PROGRAM Prg_Match
VAR
	
	boChoisirAction: BOOL;
	intChoixAction: INT;
	i: INT;
	intPrioMaxTrouvee: INT;
	boVerifPrerequis: BOOL;
	j: INT;
	intVerifAction: USINT;
	intNbActionVerifTot: INT;
	intNbActionVerifDone: INT;
	TON_1 : TON;
	boVerifPucAttente: BOOL;
	intNbPucsPris: INT;
	intNbPucDansRobot: INT;
	boGoldPris: BOOL;
	R_TRIG_StartMove: R_TRIG;
	R_TRIG_Depl: R_TRIG;
	R_TRIG_Algo: R_TRIG;
	TON_2: TON;
	R_TRIG_Move: R_TRIG;
	ADSREAD_1: ADSREAD;
	boResetExp : BOOL := TRUE;
	ADSWRITE_1: ADSWRITE;
	TON_Blink1: TON;
	TON_Blink2: TON;
	ADSWRITE_2: ADSWRITE;
	boDesactiverExp: BOOL := FALSE;;
	boEtatReset: BOOL;
	ADSREAD_2: ADSREAD;
	TON_reset: TON;
	R_TRIG_Etape: R_TRIG;
	NbPucsBalance: INT;
	bRenewDeplEv: BOOL;
	boLireEtatExp: BOOL;
	ADSREAD_3: ADSREAD;
	R_TRIG_Agold: R_TRIG;
	R_TRIG_APousser: R_TRIG;
	R_TRIG_Aok : R_TRIG;
	test: BOOL;
	attentefront: BOOL;
END_VAR

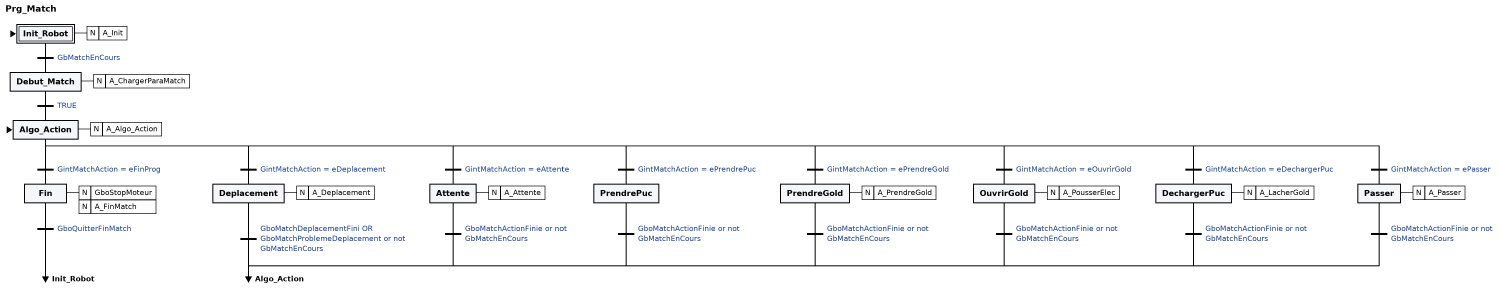
INITIAL_STEP Init_Robot:
    A_Init(N);
END_STEP
TRANSITION FROM Init_Robot TO Debut_Match
    := GbMatchEnCours;
END_TRANSITION
STEP Debut_Match:
    A_ChargerParaMatch(N);
END_STEP
TRANSITION FROM Debut_Match TO Algo_Action
    := TRUE;
END_TRANSITION
STEP Algo_Action:
    A_Algo_Action(N);
END_STEP
TRANSITION FROM Algo_Action TO Fin
    := GintMatchAction = eFinProg;
END_TRANSITION
STEP Fin:
    GboStopMoteur(N);
    A_FinMatch(N);
END_STEP
TRANSITION FROM Fin TO Init_Robot
    := GboQuitterFinMatch;
END_TRANSITION
TRANSITION FROM Algo_Action TO Deplacement
    := GintMatchAction = eDeplacement;
END_TRANSITION
STEP Deplacement:
    A_Deplacement(N);
END_STEP
TRANSITION FROM Deplacement TO Algo_Action
    := GboMatchDeplacementFini OR GboMatchProblemeDeplacement or not GbMatchEnCours;
END_TRANSITION
TRANSITION FROM Algo_Action TO Attente
    := GintMatchAction = eAttente;
END_TRANSITION
STEP Attente:
    A_Attente(N);
END_STEP
TRANSITION FROM Attente TO Algo_Action
    := GboMatchActionFinie or not GbMatchEnCours;
END_TRANSITION
TRANSITION FROM Algo_Action TO PrendrePuc
    := GintMatchAction = ePrendrePuc;
END_TRANSITION
STEP PrendrePuc:
END_STEP
TRANSITION FROM PrendrePuc TO Algo_Action
    := GboMatchActionFinie or not GbMatchEnCours;
END_TRANSITION
TRANSITION FROM Algo_Action TO PrendreGold
    := GintMatchAction = ePrendreGold;
END_TRANSITION
STEP PrendreGold:
    A_PrendreGold(N);
END_STEP
TRANSITION FROM PrendreGold TO Algo_Action
    := GboMatchActionFinie or not GbMatchEnCours;
END_TRANSITION
TRANSITION FROM Algo_Action TO OuvrirGold
    := GintMatchAction = eOuvrirGold;
END_TRANSITION
STEP OuvrirGold:
    A_PousserElec(N);
END_STEP
TRANSITION FROM OuvrirGold TO Algo_Action
    := GboMatchActionFinie or not GbMatchEnCours;
END_TRANSITION
TRANSITION FROM Algo_Action TO DechargerPuc
    := GintMatchAction = eDechargerPuc;
END_TRANSITION
STEP DechargerPuc:
    A_LacherGold(N);
END_STEP
TRANSITION FROM DechargerPuc TO Algo_Action
    := GboMatchActionFinie or not GbMatchEnCours;
END_TRANSITION
TRANSITION FROM Algo_Action TO Passer
    := GintMatchAction = ePasser;
END_TRANSITION
STEP Passer:
    A_Passer(N);
END_STEP
TRANSITION FROM Passer TO Algo_Action
    := GboMatchActionFinie or not GbMatchEnCours;
END_TRANSITION

ACTION A_Algo_Action:
R_TRIG_Algo(Clk := Algo_Action.x);

boSetPosInitiale := FALSE;

IF R_TRIG_Algo.Q THEN
	//Algorithme Action
	IF GboMatchDebutMatch THEN
		GboMatchDebutMatch := FALSE;
		boChoisirAction := TRUE;
	ELSIF GboMatchDeplacementFini THEN
		GboMatchDeplacementFini := FALSE;
		GintMatchAction := GarstMatchParaMatch[intChoixAction].uiAction;
	ELSIF GboMatchProblemeDeplacement THEN
		GboMatchProblemeDeplacement := FALSE;
		GarstMatchParaMatch[intChoixAction].boActionAttente := TRUE;
		boChoisirAction := TRUE;
	ELSIF GboMatchActionFinie THEN
	
		GboMatchActionFinie := FALSE;
		
		IF GintMatchAction <> eAttente THEN
			GarstMatchParaMatch[intChoixAction].uiNbActionFaite := GarstMatchParaMatch[intChoixAction].uiNbActionFaite + 1;	//incrmeneter le nb de fois que l'action a ete faite
			
			GNombrePointsMatch := GNombrePointsMatch + GarstMatchParaMatch[intChoixAction].intPtAction;	//increment des point de l'action qui vient d'etre aite
		
			IF GarstMatchParaMatch[intChoixAction].uiNbActionFaite >= GarstMatchParaMatch[intChoixAction].uiNbXAction AND GarstMatchParaMatch[intChoixAction].uiNbXAction <> 10 THEN
				GarstMatchParaMatch[intChoixAction].boActionDone := TRUE;
			END_IF
		END_IF
		boChoisirAction := TRUE;
		
		//Remmetre a false les action en attente
		FOR i := 1 TO GintMatchNoActionMax DO
			GarstMatchParaMatch[i].boActionAttente := FALSE;
		END_FOR
		
		
		//--------------------------------------------
		IF intChoixAction = 2 THEN
			boGoldPris := TRUE;
		END_IF
		
		IF (( 2 <= intChoixAction ) AND ( intChoixAction <= 14 )) and (GintMatchAction <> eAttente) THEN //si un pucs a ete pris, incrementer les nb de pucs dans le robot
			intNbPucDansRobot := intNbPucDansRobot + 1;
		ELSIF intChoixAction = 15 THEN	//si les pucs ont ete posé, remettre a 0 le nb de pucs dans le robot
			intNbPucDansRobot := 0;
			boGoldPris := FALSE;
		END_IF
	END_IF
	
	//-------------------------------------------------------------------------------------
	//Inserer ici moulinette algorithmique pouzr certianes actions non normales
		//Les action 28 a 30 permette de gerer quand on peut prendre / poser des pucs normaux
	//-----------------------------------------------------------------------------------------
	
	

	//------------------------------------------------------------------------------------------------
	//------------------------------------------------------------------------------------------------
	//Choix action
	
	intPrioMaxTrouvee := -1;
	
	IF boChoisirAction THEN
		boChoisirAction := FALSE;
		
		//trouver l'action la plus prioritaire possible
		FOR i := 1 TO GintMatchNoActionMax DO
			IF GarstMatchParaMatch[i].uiPrioriteAction > intPrioMaxTrouvee THEN
				//Verifier quelle peut etre faite
				IF NOT ( GarstMatchParaMatch[i].boActionDone ) AND NOT ( GarstMatchParaMatch[i].boActionAttente ) THEN
					CASE GarstMatchParaMatch[i].usiTypePrerequis OF
						0:	//Pas de prerequis
								//-> nouveau max 
							intChoixAction := i;
							intPrioMaxTrouvee := GarstMatchParaMatch[i].uiPrioriteAction;
							
						1:	//Verifier tous les prerequis
							boVerifPrerequis := TRUE;
							
							FOR j := 1 TO 15 DO
								intVerifAction := GarstMatchParaMatch[i].arusiPrerequis[j];
								IF intVerifAction <> 0 THEN
									IF NOT GarstMatchParaMatch[intVerifAction].boActionDone THEN
										boVerifPrerequis := FALSE;
									END_IF
								END_IF
							END_FOR
							
							IF boVerifPrerequis THEN
								intChoixAction := i;
								intPrioMaxTrouvee := GarstMatchParaMatch[i].uiPrioriteAction;
							END_IF
							
						2:	//Verifier si au moin un prerequis et fait
							intNbActionVerifTot := 0;
							intNbActionVerifDone := 0;
							
							FOR j := 1 TO 15 DO
								intVerifAction := GarstMatchParaMatch[i].arusiPrerequis[j];
								IF intVerifAction <> 0 THEN
										intNbActionVerifTot := intNbActionVerifTot + 1;
										IF GarstMatchParaMatch[intVerifAction].boActionDone THEN
											intNbActionVerifDone := intNbActionVerifDone + 1;
										END_IF
								END_IF							
							END_FOR
							
							IF intNbActionVerifDone >= ( intNbActionVerifTot / 2 ) THEN
								intChoixAction := i;
								intPrioMaxTrouvee := GarstMatchParaMatch[i].uiPrioriteAction;
							END_IF
							
						3:	//Verifier si tout les prerequis sont fait
							intNbActionVerifTot := 0;
							intNbActionVerifDone := 0;
							
							FOR j := 1 TO 15 DO
								intVerifAction := GarstMatchParaMatch[i].arusiPrerequis[j];
								IF intVerifAction <> 0 THEN
									intNbActionVerifTot := intNbActionVerifTot + 1;
									IF GarstMatchParaMatch[intVerifAction].boActionDone THEN
										intNbActionVerifDone := intNbActionVerifDone + 1;
									END_IF
								END_IF							
							END_FOR
							
							IF intNbActionVerifDone = intNbActionVerifTot THEN
								intChoixAction := i;
								intPrioMaxTrouvee := GarstMatchParaMatch[i].uiPrioriteAction;
							END_IF
					END_CASE
				END_IF
			END_IF
		END_FOR
		
		IF intPrioMaxTrouvee <> -1 THEN
			//action trouvée aller a la position
			GintMatchActionObjectif := intChoixAction;
			GintMatchAction := eDeplacement;
		ELSE
			//pas d'actiopn trouvée, attendre 3s
			GtimeMatchDelayAttendre := T#3S;
			GintMatchAction := eAttente;
		END_IF
	END_IF

	//Cas plus en match
	IF NOT GbMatchEnCours THEN
		GintMatchAction := eFinProg;
	END_IF
END_IF
END_ACTION

ACTION A_Attente:
TON_1(IN:= Attente.x, PT:= GtimeMatchDelayAttendre);

IF TON_1.Q THEN
	GboMatchActionFinie := true;
END_IF
END_ACTION

ACTION A_ChargerParaMatch:
IF Debut_Match.x THEN
	Fn_ViderParaMatch();

	IF GboMatchCouleur THEN
		//violet
		Fn_ChargerParaViolet();
	ELSE
		//jaune
		Fn_ChargerParaJaune();	
	END_IF
	
	GNombrePointsMatch := 5;	//5pt pose experience
	intChoixAction := 0;
	intNbPucDansRobot := 0;
	GboMatchDebutMatch := TRUE;
	boResetCommandeMoteur := FALSE;
	NbPucsBalance := 0;
	boSetPosInitiale := TRUE;
	etat_trajectoire := 1;
	StartDepl := FALSE;
	GarlrObstacles[1,2] := 0;
	GarlrObstacles[1,3] := 0;
	GboPrendreGold := FALSE;
	GboPousserElec := FALSE;
END_IF
END_ACTION

ACTION A_Deplacement:
R_TRIG_Depl(CLK:= Deplacement.x);
R_TRIG_Move(CLK := GboMoveDone);

IF  R_TRIG_Depl.Q THEN
	boReculerDepl := FALSE;
END_IF

IF R_TRIG_Depl.Q OR bRenewDeplEv THEN
	MAIN_1.pt_arrivee := GintMatchActionObjectif;
	etat_trajectoire := 2;
	bRenewDeplEv := FALSE;
	boResetCommandeMoteur := FALSE;
END_IF

R_TRIG_StartMove(CLK :=  etat_trajectoire = 10);

IF R_TRIG_StartMove.Q THEN
	//Deplacement calcul ok
	//PRG_CommandeMoteur.start_move := TRUE;	
	StartDepl := TRUE;
ELSIF etat_trajectoire = 6 THEN
	//Calcul pas ok
	GboMatchProblemeDeplacement := TRUE;
ELSIF etat_trajectoire = 7 THEN
	etat_trajectoire := 2;
ELSIF R_TRIG_Move.Q THEN
	StartDepl := FALSE;
	GboMatchDeplacementFini := TRUE;
ELSIF GbObstacleDerriere AND boSensLigneDroite AND StartDepl AND boEnLigneDroite THEN
	boEnLigneDroite := FALSE;
	boStopMotor := TRUE;
	StartDepl := FALSE;
	GarlrObstacles[1,2] := GlrPosX - 550 * COS(GlrAngle);
	GarlrObstacles[1,3] := GlrPosY - 550 * SIN(GlrAngle);
ELSIF GbObstacleDevant AND NOT boSensLigneDroite AND StartDepl AND boEnLigneDroite THEN
	boEnLigneDroite := FALSE;
	boStopMotor := TRUE;
	StartDepl := FALSE;
	GarlrObstacles[1,2] := GlrPosX + 550 * COS(GlrAngle);
	GarlrObstacles[1,3] := GlrPosY + 550 * SIN(GlrAngle);
ELSIF boStopDoneGc AND boStopDoneDr THEN
	//stop fini, refaire deplacment, reculer de 100
	boReculerDepl := TRUE;
	boStopMotor := FALSE;
	boResetCommandeMoteur := TRUE;
	bRenewDeplEv := TRUE;
END_IF
END_ACTION

ACTION A_FinMatch:
TON_2(IN:= Fin.x , PT:= T#2S);

GboMatchActionFinie := FALSE;
GboMatchDeplacementFini := FALSE;

QboEnableVentDroite := FALSE;
QboEnableVentGauche := FALSE;

GboPrendreGold := FALSE;
GboPousserElec := FALSE;

boStopMotor := TRUE;

IF TON_2.Q THEN
	boPowerMotor := FALSE;
END_IF

GstrMatchNomActionEnCour := 'Fin du match';
END_ACTION

ACTION A_Init:
R_TRIG_Etape(Clk := Init_Robot.x);

IF R_TRIG_Etape.Q THEN
	boResetExp := TRUE;
END_IF

GboQuitterFinMatch := FALSE;

IF GboMatchAuReleve THEN
	boStopMotor := FALSE;
	boPowerMotor := TRUE;
	boResetCommandeMoteur := TRUE;
ELSE
	boPowerMotor := FALSE;
END_IF

//Reset de l'experience
TON_Blink1(IN:= Init_robot.x AND NOT TON_Blink2.Q, PT:= T#1.5S);
TON_Blink2(IN:= TON_Blink1.Q, PT:= T#1.5S);

ADSREAD_2(
	NETID:= '192.168.0.151.1.1', 
	PORT:= 801, 
	IDXGRP:= 16#4020, 
	IDXOFFS:= 102, 
	LEN:= SIZEOF(boEtatReset), 
	DESTADDR:= ADR(boEtatReset), 
	READ:= TON_Blink1.Q, 
	TMOUT:= T#2S, 
	BUSY=> , 
	ERR=> , 
	ERRID=> );

ADSWRITE_1(
	NETID:= '192.168.0.151.1.1', 
	PORT:= 801, 
	IDXGRP:= 16#4020, 
	IDXOFFS:= 102, 
	LEN:= SIZEOF(boResetExp), 
	SRCADDR:= ADR(boResetExp), 
	WRITE:= TON_Blink1.Q, 
	TMOUT:= T#2S, 
	BUSY=> , 
	ERR=> , 
	ERRID=> );

ADSREAD_3(
	NETID:= '192.168.0.151.1.1', 
	PORT:= 801, 
	IDXGRP:= 16#4020, 
	IDXOFFS:= 200, 
	LEN:= SIZEOF(boLireEtatExp), 
	DESTADDR:= ADR(boLireEtatExp), 
	READ:= TON_Blink1.Q, 
	TMOUT:= T#2S, 
	BUSY=> , 
	ERR=> , 
	ERRID=> );
		
TON_reset(IN:= boEtatReset, PT:= T#4S);
IF TON_reset.Q THEN
	boResetExp := FALSE;
END_IF

IF boLireEtatExp THEN
	
	ADSWRITE_2(
		NETID:= '192.168.0.151.1.1', 
		PORT:= 801, 
		IDXGRP:= 16#4020, 
		IDXOFFS:= 100, 
		LEN:= SIZEOF(boDesactiverExp), 
		SRCADDR:= ADR(boDesactiverExp), 
		WRITE:= TON_Blink1.Q, 
		TMOUT:= T#2S, 
		BUSY=> , 
		ERR=> , 
		ERRID=> );
	
	ADSREAD_1(
		NETID:= '192.168.0.151.1.1', 
		PORT:= 801, 
		IDXGRP:= 16#4020, 
		IDXOFFS:= 200, 
		LEN:= SIZEOF(Prog_Activer_Experience.boLireEtatExp), 
		DESTADDR:= ADR(Prog_Activer_Experience.boLireEtatExp), 
		READ:= TON_Blink1.Q, 
		TMOUT:= T#2S, 
		BUSY=> , 
		ERR=> , 
		ERRID=> );
		
END_IF
END_ACTION

ACTION A_LacherGold:
QboEnableVentDroite := FALSE;
QboEnableVentGauche := FALSE;

GboMatchActionFinie := TRUE;
END_ACTION

ACTION A_Passer:
GboMatchActionFinie := TRUE;
END_ACTION

ACTION A_PousserElec:
R_TRIG_APousser( Clk := OuvrirGold.x );

IF R_TRIG_APousser.Q THEN
	GboPousserElec := TRUE;
	IF GboActionok THEN
		attentefront := TRUE;
	ELSE
		attentefront := FALSE;
	END_IF
END_IF

IF NOT GboActionok THEN
	attentefront := FALSE;
END_IF

IF (NOT attentefront) AND GboActionok THEN
	GboPousserElec := FALSE;
	GboMatchActionFinie := TRUE;
END_IF
END_ACTION

ACTION A_PrendreGold:
R_TRIG_Agold( Clk := PrendreGold.x );

IF R_TRIG_Agold.Q THEN
	GboPrendreGold := TRUE;
		IF GboActionok THEN
		attentefront := TRUE;
	ELSE
		attentefront := FALSE;
	END_IF
END_IF

IF NOT GboActionok THEN
	attentefront := FALSE;
END_IF

IF (NOT attentefront) AND GboActionok THEN
	GboPrendreGold := FALSE;
	GboMatchActionFinie := TRUE;
END_IF
END_ACTION

END_PROGRAM

(* stored: Version 1.1.0.1, ProductVersion 3.1.4022.18
   POU Prg_Match: Id {9b37f1e8-f8c1-4599-bd45-92a36110e6ae}, SpecialFunc None
   Action A_Algo_Action: Id {a05a9753-ab2e-453f-864d-c300a9574544}
   Action A_Attente: Id {e8037cf4-7f39-4e74-832d-4245ef3e85d6}
   Action A_ChargerParaMatch: Id {f78661cb-0b7b-4075-a7f9-0224dd77acd4}
   Action A_Deplacement: Id {a9eeb879-a394-441d-b4d8-781b6cfbfa13}
   Action A_FinMatch: Id {91d0a8af-c7fe-444b-9e91-b54f5e28bfee}
   Action A_Init: Id {374d6e26-ad63-4bc5-b31e-414496d10915}
   Action A_LacherGold: Id {ddf45cf6-d570-498b-aca9-59a85195f0e6}
   Action A_Passer: Id {276ef024-6ae4-4f46-97ec-5e04ef4c5061}
   Action A_PousserElec: Id {48edcd21-d0f4-4a08-9a22-2467c43f1094}
   Action A_PrendreGold: Id {3cae239a-0cbb-4b25-87b9-ebc3ff4746d0} *)
